Fanuc KAREL source: kb00002.KL

-- PROVISIONAL review KL for V940-1; original PC SHA256 92a58b4495d3026f95b427fec1557fffe6a2c2a5d2e8939130d75976bcbb8a53
-- Incomplete behavior may be omitted. Consult companion uncertainty JSON. Do not deploy.
PROGRAM KB00002
%NOLOCKGROUP
VAR
  P1 : INTEGER
  RESULT : INTEGER
BEGIN
  -- V9_ZERO_TABLE_METADATA_HINT layout=0001; no indexed target words; source/name/runtime held
  -- UNRESOLVED_PC offsets 5-12; opcodes 9D,23
  -- UNRESOLVED_PC offsets 17-30; opcodes 21,50,23
  -- UNRESOLVED_PC offsets 35-39; opcodes 7F
END KB00002
